Staubli VAL3: clkDoAirex.pgx

program clkDoAirex()
begin
  bDoAirex=true
end
